KUKA KRL program: wkz_off_st_geo.src, wkz_off_st_geo.dat

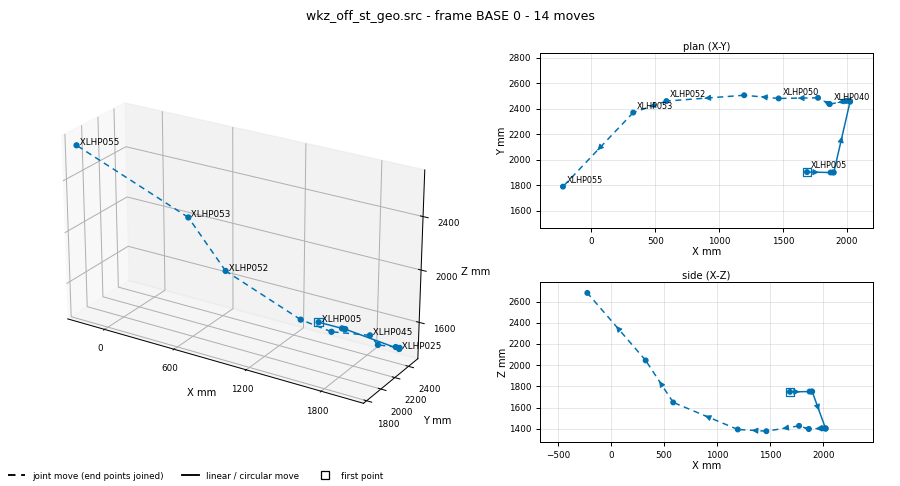
[picture p0: tool path of wkz_off_st_geo.src in frame BASE 0, 14 of 14 moves have a stored position in this frame; points joined in program order, loops and branches not executed]
--- wkz_off_st_geo.src ---
&ACCESS RVO2
&REL 409
&COMMENT Retira Gripper Geo
&PARAM DISKPATH = KRC:\R1\Program
DEF wkz_off_st_geo( )
;FOLD INI
   ;FOLD BASISTECH INI
      GLOBAL INTERRUPT DECL 3 WHEN $STOPMESS==TRUE DO IR_STOPM ( )
      INTERRUPT ON 3
      BAS (#INITMOV,0 )
   ;ENDFOLD (BASISTECH INI)
   ;FOLD SPOTTECH INI
      USERSPOT(#INIT)
   ;ENDFOLD (SPOTTECH INI)
   ;FOLD GRIPPERTECH INI
      USER_GRP(0,DUMMY,DUMMY,GDEFAULT)
   ;ENDFOLD (GRIPPERTECH INI)
   ;FOLD USER INI
      ;Make your modifications here

   ;ENDFOLD (USER INI)
;ENDFOLD (INI)

; Estacao P13.060 - Robo R1
; Programa: Pega Gripper Garra
; Accelo na Geobox. Gripper F5_6500_0026_656
; Caracterização dos meios de produção:
; 02/09/2014 09:15 Changes by KUKA Roboter do Brasil

chk_w8_wechs_ok ( )   ; CHECK FERRAMENTA: TOOL CHANGER

;FOLD OUT 3337 'R1_Retira Garra Geo' State=TRUE ;%{PE}%R 8.2.20,%MKUKATPBASIS,%COUT,%VOUTX,%P 2:3337, 3:R1_Retira Garra Geo, 5:TRUE, 6:
$OUT[3337]=TRUE
;ENDFOLD
;FOLD WAIT FOR ( IN 3337 'R1_Aguarda Lib. Entrar Geo' );%{PE}%R 8.2.20,%MKUKATPBASIS,%CEXT_WAIT_FOR,%VEXT_WAIT_FOR,%P 2:, 4:, 5:$IN, 6:3337, 7:R1_Aguarda Lib. Entrar Geo, 9:
WAIT FOR  ( $IN[3337] )
;ENDFOLD
;FOLD OUT 3337 'R1_Retira Garra Geo' State=FALSE ;%{PE}%R 8.2.20,%MKUKATPBASIS,%COUT,%VOUTX,%P 2:3337, 3:R1_Retira Garra Geo, 5:FALSE, 6:
$OUT[3337]=FALSE
;ENDFOLD
;FOLD OUT 3346 'R1_Entrega Peca Geo' State=FALSE ;%{PE}%R 8.2.20,%MKUKATPBASIS,%COUT,%VOUTX,%P 2:3346, 3:R1_Entrega Peca Geo, 5:FALSE, 6:
$OUT[3346]=FALSE
;ENDFOLD
;FOLD OUT 3343 'R1_Entregou Peca Geo' State=FALSE ;%{PE}%R 8.2.20,%MKUKATPBASIS,%COUT,%VOUTX,%P 2:3343, 3:R1_Entregou Peca Geo, 5:FALSE, 6:
$OUT[3343]=FALSE
;ENDFOLD

;FOLD OUT 3369 'Area de Solda' State=FALSE ;%{PE}%R 8.2.20,%MKUKATPBASIS,%COUT,%VOUTX,%P 2:3369, 3:Area de Solda, 5:FALSE, 6:
$OUT[3369]=FALSE
;ENDFOLD

;FOLD Kollision.Ueberwachung_3_Ein ;%{PE}%MKUKATPUSER
COLLSTOP( 3, 1 ) ;INTERRUPTUEBERWACHT
;ENDFOLD

;FOLD PTP LHP005 CONT Vel=60 % PDAT3 Tool[2]:Gripper Lat Esq Accelo Base[0];%{PE}%R 4.1.15,%MKUKATPBASIS,%CMOVE,%VPTP,%P 1:PTP, 2:LHP005, 3:C_PTP, 5:60, 7:PDAT3
$BWDSTART=FALSE
PDAT_ACT=PPDAT3
BAS (#PTP_DAT )
FDAT_ACT=FLHP005
BAS (#FRAMES )
BAS (#VEL_PTP,60 )
PTP  XLHP005 C_PTP
;ENDFOLD

;FOLD OUT 224 'Bloqueio MPS'  State= FALSE ;%{PE}%R 4.1.16,%MKUKATPBASIS,%COUT,%VOUTX,%P 2:224, 3:'Bloqueio MPS', 5:FALSE, 6:
$OUT[224]=FALSE
;ENDFOLD
;FOLD OUT 223 'Desbloqueio MPS'  State= TRUE ;%{PE}%R 4.1.16,%MKUKATPBASIS,%COUT,%VOUTX,%P 2:223, 3:'Desbloqueio MPS', 5:TRUE, 6:
$OUT[223]=TRUE
;ENDFOLD

;FOLD LIN LHP010 Vel=0.3 m/s CPDAT11 Tool[8]:Tool Changer Base[0];%{PE}%R 8.2.20,%MKUKATPBASIS,%CMOVE,%VLIN,%P 1:LIN, 2:LHP010, 3:, 5:0.3, 7:CPDAT11
$BWDSTART=FALSE
LDAT_ACT=LCPDAT11
FDAT_ACT=FLHP010
BAS(#CP_PARAMS,0.3)
LIN XLHP010
;ENDFOLD

;FOLD WAIT FOR IN 217 'MPS destravado'  State= TRUE ;%{PE}%R 4.1.16,%MKUKATPBASIS,%CWAIT_FOR,%VWAIT_FOR,%P 1:0, 2:217, 3:'MPS destravado', 5:TRUE, 6:
WAIT FOR $IN[217]==TRUE
;ENDFOLD
;FOLD WAIT FOR IN 221 'MPS travado'  State= FALSE ;%{PE}%R 4.1.16,%MKUKATPBASIS,%CWAIT_FOR,%VWAIT_FOR,%P 1:0, 2:221, 3:'MPS travado', 5:FALSE, 6:
WAIT FOR $IN[221]==FALSE
;ENDFOLD

;FOLD LIN LHP015 Vel=0.25 m/s CPDAT12 Tool[8]:Tool Changer Base[0];%{PE}%R 8.2.20,%MKUKATPBASIS,%CMOVE,%VLIN,%P 1:LIN, 2:LHP015, 3:, 5:0.25, 7:CPDAT12
$BWDSTART=FALSE
LDAT_ACT=LCPDAT12
FDAT_ACT=FLHP015
BAS(#CP_PARAMS,0.25)
LIN XLHP015
;ENDFOLD

;FOLD ;  posicao de pega do gripper;%{PE}%R 4.1.16,%MKUKATPBASIS,%CCOMMENT,%VNORMAL,%P 2: posicao de pega do gripper
;ENDFOLD
;FOLD LIN LHP020  Vel= 0.25 m/s CPDAT15 Tool[8]:Tool Changer Base[0];%{PE}%R 4.1.16,%MKUKATPBASIS,%CMOVE,%VLIN,%P 1:LIN, 2:LHP020, 3:, 5:0.25, 7:CPDAT15
$BWDSTART = FALSE
LDAT_ACT=LCPDAT15
BAS(#CP_DAT)
FDAT_ACT=FLHP020
BAS(#FRAMES)
BAS(#VEL_CP,0.25)
LIN XLHP020
;ENDFOLD

;FOLD WAIT Time= 1 sec;%{PE}%R 4.1.16,%MKUKATPBASIS,%CWAIT,%VWAIT,%P 2:1
WAIT SEC 1
;ENDFOLD
;FOLD WAIT FOR IN 219 'placas de suporte fundidas'  State= TRUE ;%{PE}%R 4.1.16,%MKUKATPBASIS,%CWAIT_FOR,%VWAIT_FOR,%P 1:0, 2:219, 3:'placas de suporte fundidas', 5:TRUE, 6:
WAIT FOR $IN[219]==TRUE
;ENDFOLD
;FOLD IBUS  OFF;%{PE}%R 4.1.16,%MKUKATPBASIS,%CIBUS,%VMAP,%P 2:#OFF, 3:1
$IBUS_OFF=$IBUS_ON
$IBUS_ON=0
;ENDFOLD
;FOLD OUT 223 'Desbloqueio MPS'  State= FALSE ;%{PE}%R 4.1.16,%MKUKATPBASIS,%COUT,%VOUTX,%P 2:223, 3:'Desbloqueio MPS', 5:FALSE, 6:
$OUT[223]=FALSE
;ENDFOLD
;FOLD OUT 224 'Bloqueio MPS'  State= TRUE ;%{PE}%R 4.1.16,%MKUKATPBASIS,%COUT,%VOUTX,%P 2:224, 3:'Bloqueio MPS', 5:TRUE, 6:
$OUT[224]=TRUE
;ENDFOLD
;FOLD WAIT FOR IN 217 'MPS destravado'  State= FALSE ;%{PE}%R 4.1.16,%MKUKATPBASIS,%CWAIT_FOR,%VWAIT_FOR,%P 1:0, 2:217, 3:'MPS destravado', 5:FALSE, 6:
WAIT FOR $IN[217]==FALSE
;ENDFOLD
;FOLD WAIT FOR IN 221 'MPS travado'  State= TRUE ;%{PE}%R 4.1.16,%MKUKATPBASIS,%CWAIT_FOR,%VWAIT_FOR,%P 1:0, 2:221, 3:'MPS travado', 5:TRUE, 6:
WAIT FOR $IN[221]==TRUE
;ENDFOLD
;FOLD IBUS  ON SEGMENT_2;%{PE}%R 4.1.16,%MKUKATPBASIS,%CIBUS,%VMAP,%P 2:#ON, 3:2
$IBUS_ON=IBUS_SEGMENT[2]
$IBUS_OFF=0
;ENDFOLD
;FOLD WAIT Time= 1 sec;%{PE}%R 4.1.16,%MKUKATPBASIS,%CWAIT,%VWAIT,%P 2:1
WAIT SEC 1
;ENDFOLD

;FOLD OUT 3366 'R1_Solicita Sair com Garra' State=TRUE ;%{PE}%R 8.2.20,%MKUKATPBASIS,%COUT,%VOUTX,%P 2:3366, 3:R1_Solicita Sair com Garra, 5:TRUE, 6:
$OUT[3366]=TRUE
;ENDFOLD
;FOLD WAIT FOR ( IN 3335 'R1_Aguarda Lib. Retirar Garra' );%{PE}%R 8.2.20,%MKUKATPBASIS,%CEXT_WAIT_FOR,%VEXT_WAIT_FOR,%P 2:, 4:, 5:$IN, 6:3335, 7:R1_Aguarda Lib. Retirar Garra, 9:
WAIT FOR  ( $IN[3335] )
;ENDFOLD
;FOLD OUT 3366 'R1_Solicita Sair com Garra' State=FALSE ;%{PE}%R 8.2.20,%MKUKATPBASIS,%COUT,%VOUTX,%P 2:3366, 3:R1_Solicita Sair com Garra, 5:FALSE, 6:
$OUT[3366]=FALSE
;ENDFOLD

;FOLD SET GRP 1  State= OPN  GDAT1;%{PE}%R 4.1.7,%MKUKATPGRP,%CGRP,%VGRP,%P 2:1, 4:1, 5:#NO, 6:GDAT1, 8:0, 10:0
H50(GRP,1,1,GGDAT1)
;ENDFOLD
chk_grp1_opn ( )
;FOLD OUT 4 'Liga Vacuo' State=FALSE ;%{PE}%R 8.2.20,%MKUKATPBASIS,%COUT,%VOUTX,%P 2:4, 3:Liga Vacuo, 5:FALSE, 6:
$OUT[4]=FALSE
;ENDFOLD
;FOLD PULSE 3 'Sopro' State=TRUE Time=2 sec;%{PE}%R 8.2.20,%MKUKATPBASIS,%COUT,%VPULSE,%P 2:3, 3:Sopro, 5:TRUE, 6:, 8:2
PULSE($OUT[3], TRUE,2)
;ENDFOLD
;FOLD PULSE 3335 'R1_Retirou Garra Geo' State=TRUE CONT Time=3 sec;%{PE}%R 8.2.20,%MKUKATPBASIS,%COUT,%VPULSE,%P 2:3335, 3:R1_Retirou Garra Geo, 5:TRUE, 6:CONTINUE, 8:3
CONTINUE
PULSE($OUT[3335], TRUE,3)
;ENDFOLD
;FOLD OUT 3369 'Area de Solda' State=TRUE ;%{PE}%R 8.2.20,%MKUKATPBASIS,%COUT,%VOUTX,%P 2:3369, 3:Area de Solda, 5:TRUE, 6:
$OUT[3369]=TRUE
;ENDFOLD

;FOLD LIN LHP025 CONT Vel= 0.2 m/s CPDAT5 Tool[2]:Gripper Lat Esq Accelo Base[0];%{PE}%R 4.1.16,%MKUKATPBASIS,%CMOVE,%VLIN,%P 1:LIN, 2:LHP025, 3:C_DIS, 5:0.2, 7:CPDAT5
$BWDSTART = FALSE
LDAT_ACT=LCPDAT5
BAS(#CP_DAT)
FDAT_ACT=FLHP025
BAS(#FRAMES)
BAS(#VEL_CP,0.2)
LIN XLHP025 C_DIS
;ENDFOLD
;FOLD LIN LHP030 CONT Vel= 0.3 m/s CPDAT3 Tool[2]:Gripper Lat Esq Accelo Base[0];%{PE}%R 4.1.16,%MKUKATPBASIS,%CMOVE,%VLIN,%P 1:LIN, 2:LHP030, 3:C_DIS, 5:0.3, 7:CPDAT3
$BWDSTART = FALSE
LDAT_ACT=LCPDAT3
BAS(#CP_DAT)
FDAT_ACT=FLHP030
BAS(#FRAMES)
BAS(#VEL_CP,0.3)
LIN XLHP030 C_DIS
;ENDFOLD

;FOLD LIN LHP035 CONT Vel=2 m/s CPDAT4 Tool[2]:Gripper Lat Esq Accelo Base[0];%{PE}%R 8.2.20,%MKUKATPBASIS,%CMOVE,%VLIN,%P 1:LIN, 2:LHP035, 3:C_DIS C_DIS, 5:2, 7:CPDAT4
$BWDSTART=FALSE
LDAT_ACT=LCPDAT4
FDAT_ACT=FLHP035
BAS(#CP_PARAMS,2)
LIN XLHP035 C_DIS C_DIS
;ENDFOLD
;FOLD WAIT FOR IN 219 'placas de suporte fundidas'  State= TRUE ;%{PE}%R 4.1.16,%MKUKATPBASIS,%CWAIT_FOR,%VWAIT_FOR,%P 1:0, 2:219, 3:'placas de suporte fundidas', 5:TRUE, 6:
WAIT FOR $IN[219]==TRUE
;ENDFOLD

;FOLD PTP LHP040 CONT Vel= 60 % P_OLP4 Tool[2]:Gripper Lat Esq Accelo Base[0];%{PE}%R 4.1.16,%MKUKATPBASIS,%CMOVE,%VPTP,%P 1:PTP, 2:LHP040, 3:C_PTP, 5:60, 7:P_OLP4
$BWDSTART = FALSE
PDAT_ACT=PP_OLP4
BAS(#PTP_DAT)
FDAT_ACT=FLHP040
BAS(#FRAMES)
BAS(#VEL_PTP,60)
PTP XLHP040 C_PTP
;ENDFOLD
;FOLD PTP LHP045 CONT Vel= 50 % PDAT26 Tool[2]:Gripper Lat Esq Accelo Base[0];%{PE}%R 4.1.16,%MKUKATPBASIS,%CMOVE,%VPTP,%P 1:PTP, 2:LHP045, 3:C_PTP, 5:50, 7:PDAT26
$BWDSTART = FALSE
PDAT_ACT=PPDAT26
BAS(#PTP_DAT)
FDAT_ACT=FLHP045
BAS(#FRAMES)
BAS(#VEL_PTP,50)
PTP XLHP045 C_PTP
;ENDFOLD
;FOLD PTP LHP050 CONT Vel=60 % PDAT11 Tool[2]:Gripper Lat Esq Accelo Base[0];%{PE}%R 8.2.20,%MKUKATPBASIS,%CMOVE,%VPTP,%P 1:PTP, 2:LHP050, 3:C_DIS, 5:60, 7:PDAT11
$BWDSTART=FALSE
PDAT_ACT=PPDAT11
FDAT_ACT=FLHP050
BAS(#PTP_PARAMS,60)
PTP XLHP050 C_DIS
;ENDFOLD
;FOLD PTP LHP051 CONT Vel=60 % PDAT7 Tool[2]:Gripper Lat Esq Accelo Base[0];%{PE}%R 8.2.20,%MKUKATPBASIS,%CMOVE,%VPTP,%P 1:PTP, 2:LHP051, 3:C_DIS, 5:60, 7:PDAT7
$BWDSTART=FALSE
PDAT_ACT=PPDAT7
FDAT_ACT=FLHP051
BAS(#PTP_PARAMS,60)
PTP XLHP051 C_DIS
;ENDFOLD
;FOLD PTP LHP052 CONT Vel=60 % PDAT10 Tool[2]:Gripper Lat Esq Accelo Base[0];%{PE}%R 8.2.20,%MKUKATPBASIS,%CMOVE,%VPTP,%P 1:PTP, 2:LHP052, 3:C_DIS, 5:60, 7:PDAT10
$BWDSTART=FALSE
PDAT_ACT=PPDAT10
FDAT_ACT=FLHP052
BAS(#PTP_PARAMS,60)
PTP XLHP052 C_DIS
;ENDFOLD
;FOLD PTP LHP053 CONT Vel=60 % PDAT9 Tool[2]:Gripper Lat Esq Accelo Base[0];%{PE}%R 8.2.20,%MKUKATPBASIS,%CMOVE,%VPTP,%P 1:PTP, 2:LHP053, 3:C_DIS, 5:60, 7:PDAT9
$BWDSTART=FALSE
PDAT_ACT=PPDAT9
FDAT_ACT=FLHP053
BAS(#PTP_PARAMS,60)
PTP XLHP053 C_DIS
;ENDFOLD
;FOLD PTP LHP055 CONT Vel=50 % PDAT22 Tool[2]:Gripper Lat Esq Accelo Base[0];%{PE}%R 8.2.20,%MKUKATPBASIS,%CMOVE,%VPTP,%P 1:PTP, 2:LHP055, 3:C_DIS, 5:50, 7:PDAT22
$BWDSTART=FALSE
PDAT_ACT=PPDAT22
FDAT_ACT=FLHP055
BAS(#PTP_PARAMS,50)
PTP XLHP055 C_DIS
;ENDFOLD

;FOLD OUT 3337 'R1_Retira Garra Geo' State=TRUE CONT;%{PE}%R 8.2.20,%MKUKATPBASIS,%COUT,%VOUTX,%P 2:3337, 3:R1_Retira Garra Geo, 5:TRUE, 6:CONTINUE
CONTINUE
$OUT[3337]=TRUE
;ENDFOLD

END

--- wkz_off_st_geo.dat ---
&ACCESS RVO2
&REL 409
&COMMENT Retira Gripper Geo
&PARAM DISKPATH = KRC:\R1\Program
DEFDAT  wkz_off_st_geo
;FOLD EXTERNAL DECLARATIONS;%{PE}%MKUKATPBASIS,%CEXT,%VCOMMON,%P
;FOLD GRIPPERTECH EXT
EXT  H50 (INT  :IN,INT  :IN,INT  :IN,GRP_TYP  :IN )
;ENDFOLD (GRIPPERTECH EXT)
;FOLD SPOTTECH EXT
EXT  USERSPOT (S_COMMAND  :IN,SPOT_TYPE  :IN )
;ENDFOLD (SPOTTECH EXT)
;FOLD BASISTECH EXT;%{PE}%MKUKATPBASIS,%CEXT,%VEXT,%P
EXT  BAS (BAS_COMMAND  :IN,REAL  :IN )
DECL INT SUCCESS
;ENDFOLD (BASISTECH EXT)
;FOLD USER EXT;%{E}%MKUKATPUSER,%CEXT,%VEXT,%P
;Make your modifications here

;ENDFOLD (USER EXT)
;ENDFOLD (EXTERNAL DECLARATIONS)

;# ============ START PATH : ba_p13060r1_ltc_01 =============
DECL FDAT FLHP020={TOOL_NO 8,BASE_NO 0,IPO_FRAME #BASE}
DECL E6POS XLHP020={X 1896.38098,Y 1901.17798,Z 1752.06396,A -85.0355911,B 75.0925217,C -86.0191422,S 18,T 35,E1 0.0,E2 0.0,E3 0.0,E4 0.0,E5 0.0,E6 0.0}
DECL FDAT Fp4={TOOL_NO 2,BASE_NO 0,IPO_FRAME #BASE}
DECL E6POS Xp4={X 1992.50098,Y 2460.31396,Z 1405.73596,A -89.0228882,B 0.185930401,C -89.5983276,S 2,T 35,E1 0.0,E2 0.0,E3 0.0,E4 0.0,E5 0.0,E6 0.0}
DECL LDAT LL_OLP2={VEL 0.25,ACC 90.0,APO_DIST 2.0,APO_FAC 0.0}
DECL FDAT FLHP040={TOOL_NO 2,BASE_NO 0,IPO_FRAME #BASE}
DECL PDAT PP_OLP4={VEL 100.0,ACC 90.0,APO_DIST 30.0}
DECL E6POS XLHP040={X 1864.59302,Y 2435.71997,Z 1398.99194,A -89.3946533,B 0.327209085,C -89.8916321,S 18,T 35,E1 0.0,E2 0.0,E3 0.0,E4 0.0,E5 0.0,E6 0.0}
DECL PDAT PPDAT3={VEL 60.0,ACC 85.0,APO_DIST 30.0}
DECL PDAT PPDAT4={VEL 100.0,ACC 90.0,APO_DIST 30.0,APO_MODE #CDIS}
DECL E6POS XLHP045={X 1772.84998,Y 2485.021,Z 1428.75696,A -89.6036911,B 5.70348883,C -90.1840286,S 18,T 35,E1 0.0,E2 0.0,E3 0.0,E4 0.0,E5 0.0,E6 0.0}
DECL FDAT FLHP045={TOOL_NO 2,BASE_NO 0,IPO_FRAME #BASE}
DECL E6POS XLHP050={X 1464.948,Y 2480.08301,Z 1378.42798,A -86.6316299,B 5.11988878,C -98.4016876,S 18,T 35,E1 0.0,E2 0.0,E3 0.0,E4 0.0,E5 0.0,E6 0.0}
DECL FDAT FLHP050={TOOL_NO 2,BASE_NO 0,IPO_FRAME #BASE}
DECL LDAT LCPDAT2={VEL 2.0,ACC 85.0,APO_DIST 20.0,APO_FAC 50.0}
DECL GRP_SUGG_T LAST_GRP={NUMBER[] "1                       ",STATE[] "1                       ",PARAMS[] "GDAT1                   "}
DECL GRP_TYP GGDAT1={G_APO #NO,GRP_TIME 0.200000003,CTRL #OFF,DLY 0,DST 1}
DECL E6POS XLHP025={X 2023.43896,Y 2454.15991,Z 1401.18994,A -89.1424637,B 0.328501195,C -89.5951538,S 18,T 35,E1 0.0,E2 0.0,E3 0.0,E4 0.0,E5 0.0,E6 0.0}
DECL FDAT FLHP025={TOOL_NO 2,BASE_NO 0,IPO_FRAME #BASE}
DECL LDAT LCPDAT5={VEL 2.0,ACC 100.0,APO_DIST 2.0,APO_FAC 50.0}
DECL E6POS XLHP030={X 2022.849,Y 2460.35303,Z 1406.90601,A -89.0257721,B 0.139669403,C -89.5021896,S 2,T 35,E1 0.0,E2 0.0,E3 0.0,E4 0.0,E5 0.0,E6 0.0}
DECL FDAT FLHP030={TOOL_NO 2,BASE_NO 0,IPO_FRAME #BASE}
DECL LDAT LCPDAT3={VEL 2.0,ACC 90.0,APO_DIST 2.0,APO_FAC 50.0}
DECL LDAT LCPDAT11={VEL 2.0,ACC 90.0,APO_DIST 100.0,APO_FAC 50.0}
DECL E6POS XLHP010={X 1871.48401,Y 1900.80396,Z 1751.72095,A -85.027832,B 75.0897369,C -86.0116425,S 18,T 35,E1 0.0,E2 0.0,E3 0.0,E4 0.0,E5 0.0,E6 0.0}
DECL FDAT FLHP010={TOOL_NO 8,BASE_NO 0,IPO_FRAME #BASE,TQ_STATE FALSE}
DECL E6POS XLHP055={X -221.914398,Y 1790.33997,Z 2680.93799,A -84.7821732,B 77.6812134,C -170.099701,S 18,T 43,E1 0.0,E2 0.0,E3 0.0,E4 0.0,E5 0.0,E6 0.0}
DECL FDAT FLHP055={TOOL_NO 2,BASE_NO 0,IPO_FRAME #BASE,TQ_STATE FALSE}
DECL PDAT PPDAT22={VEL 100.0,ACC 100.0,APO_DIST 10.0,APO_MODE #CDIS}
DECL LDAT LCPDAT12={VEL 2.0,ACC 75.0,APO_DIST 5.0,APO_FAC 50.0}
DECL PDAT PPDAT26={VEL 100.0,ACC 85.0,APO_DIST 30.0}
DECL E6POS XLHP015={X 1891.69495,Y 1901.10095,Z 1751.979,A -85.0317917,B 75.0909805,C -86.0155106,S 18,T 35,E1 0.0,E2 0.0,E3 0.0,E4 0.0,E5 0.0,E6 0.0}
DECL FDAT FLHP015={TOOL_NO 8,BASE_NO 0,IPO_FRAME #BASE,TQ_STATE FALSE}
DECL LDAT LCPDAT15={VEL 2.0,ACC 90.0,APO_DIST 100.0,APO_FAC 50.0}
DECL E6POS XLHP005={X 1686.87598,Y 1904.25806,Z 1748.90906,A -86.3585892,B 75.039093,C -87.1308594,S 2,T 35,E1 0.0,E2 0.0,E3 0.0,E4 0.0,E5 0.0,E6 0.0}
DECL FDAT FLHP005={TOOL_NO 8,BASE_NO 0,IPO_FRAME #BASE}
DECL BASIS_SUGG_T LAST_BASIS={POINT1[] "LHP052                  ",POINT2[] "LHP052                  ",CP_PARAMS[] "CPDAT0                  ",PTP_PARAMS[] "PDAT10                  ",CONT[] "                        ",CP_VEL[] "0.3                     ",PTP_VEL[] "60                      ",SYNC_PARAMS[] "SYNCDAT                 ",SPL_NAME[] "S0                      "}
DECL E6POS XLHP026={X 1779.83301,Y 2450.62012,Z 1399.65796,A -89.1403503,B 0.323707789,C -89.5841599,S 18,T 35,E1 0.0,E2 0.0,E3 0.0,E4 0.0,E5 0.0,E6 0.0}
DECL FDAT FLHP026={TOOL_NO 2,BASE_NO 0,IPO_FRAME #BASE,POINT2[] " ",TQ_STATE FALSE}
DECL LDAT LCPDAT1={VEL 2.0,ACC 100.0,APO_DIST 100.0,APO_FAC 50.0,AXIS_VEL 100.0,AXIS_ACC 100.0,ORI_TYP #VAR,CIRC_TYP #BASE,JERK_FAC 50.0,GEAR_JERK 50.0,EXAX_IGN 0}
DECL E6POS XLHP027={X 1762.18298,Y 2450.34692,Z 1381.23499,A -89.1904221,B 0.385173112,C -96.4581909,S 18,T 35,E1 0.0,E2 0.0,E3 0.0,E4 0.0,E5 0.0,E6 0.0}
DECL FDAT FLHP027={TOOL_NO 2,BASE_NO 0,IPO_FRAME #BASE,POINT2[] " ",TQ_STATE FALSE}
DECL PDAT PPDAT1={VEL 100.0,ACC 90.0,APO_DIST 100.0,GEAR_JERK 50.0}
DECL E6POS XLHP028={X 1762.04395,Y 2404.74902,Z 1375.10303,A -89.1892166,B 0.401495486,C -96.4518967,S 18,T 35,E1 0.0,E2 0.0,E3 0.0,E4 0.0,E5 0.0,E6 0.0}
DECL FDAT FLHP028={TOOL_NO 2,BASE_NO 0,IPO_FRAME #BASE,POINT2[] " ",TQ_STATE FALSE}
DECL PDAT PPDAT2={VEL 100.0,ACC 90.0,APO_DIST 100.0,GEAR_JERK 50.0}
DECL E6POS XLHP029={X 1651.26294,Y 2403.11597,Z 1374.71399,A -89.1894836,B 0.401636302,C -96.4478073,S 18,T 35,E1 0.0,E2 0.0,E3 0.0,E4 0.0,E5 0.0,E6 0.0}
DECL FDAT FLHP029={TOOL_NO 2,BASE_NO 0,IPO_FRAME #BASE,POINT2[] " ",TQ_STATE FALSE}
DECL PDAT PPDAT5={VEL 100.0,ACC 90.0,APO_DIST 100.0,GEAR_JERK 50.0}
DECL FDAT FLHP035={TOOL_NO 2,BASE_NO 0,IPO_FRAME #BASE,POINT2[] " ",TQ_STATE FALSE}
DECL E6POS XLHP035={X 1992.49902,Y 2460.31299,Z 1405.73401,A -89.0231323,B 0.186079606,C -89.5979233,S 18,T 35,E1 0.0,E2 0.0,E3 0.0,E4 0.0,E5 0.0,E6 0.0}
DECL LDAT LCPDAT4={VEL 2.0,ACC 90.0,APO_DIST 2.0,APO_FAC 50.0,AXIS_VEL 100.0,AXIS_ACC 100.0,ORI_TYP #VAR,CIRC_TYP #BASE,JERK_FAC 50.0,GEAR_JERK 50.0,EXAX_IGN 0}
DECL SPOT_SUGG_T LAST_SPOT={GUN[] " 1                      ",RETR_CMD[] "#OPN                    ",CHOISE[] "#FIRST                  ",CLO_TM[] "0                       ",PGNO1[] " 1                      ",PRESS1[] "0                       ",PGNO2[] " 1                      ",PRESS2[] "0                       ",SPOT_PARAMS[] "NORMAL                  "}
DECL E6POS XLHP036={X 1788.44397,Y 2466.40698,Z 1395.04797,A -89.6003494,B 0.3782776,C -89.9430923,S 18,T 35,E1 0.0,E2 0.0,E3 0.0,E4 0.0,E5 0.0,E6 0.0}
DECL FDAT FLHP036={TOOL_NO 2,BASE_NO 0,IPO_FRAME #BASE,POINT2[] " ",TQ_STATE FALSE}
DECL PDAT PPDAT6={VEL 100.0,ACC 90.0,APO_DIST 30.0,APO_MODE #CDIS,GEAR_JERK 50.0}
DECL LDAT LCPDAT6={VEL 2.0,ACC 90.0,APO_DIST 2.0,APO_FAC 50.0,AXIS_VEL 100.0,AXIS_ACC 100.0,ORI_TYP #VAR,CIRC_TYP #BASE,JERK_FAC 50.0,GEAR_JERK 50.0,EXAX_IGN 0}
DECL E6POS XLHP051={X 1195.36304,Y 2505.11108,Z 1394.828,A -83.3905563,B 11.3238802,C -106.139702,S 18,T 35,E1 0.0,E2 0.0,E3 0.0,E4 0.0,E5 0.0,E6 0.0}
DECL FDAT FLHP051={TOOL_NO 2,BASE_NO 0,IPO_FRAME #BASE,POINT2[] " ",TQ_STATE FALSE}
DECL PDAT PPDAT7={VEL 100.0,ACC 85.0,APO_DIST 100.0,APO_MODE #CDIS,GEAR_JERK 50.0}
DECL E6POS XLHP054={X 327.607391,Y 2369.56299,Z 2045.41394,A -78.953537,B 42.0104408,C -130.848007,S 18,T 35,E1 0.0,E2 0.0,E3 0.0,E4 0.0,E5 0.0,E6 0.0}
DECL FDAT FLHP054={TOOL_NO 2,BASE_NO 0,IPO_FRAME #BASE,POINT2[] " ",TQ_STATE FALSE}
DECL PDAT PPDAT8={VEL 100.0,ACC 85.0,APO_DIST 100.0,GEAR_JERK 50.0}
DECL E6POS XLHP053={X 327.606293,Y 2369.56494,Z 2045.42297,A -78.9541473,B 42.0112991,C -130.848801,S 18,T 35,E1 0.0,E2 0.0,E3 0.0,E4 0.0,E5 0.0,E6 0.0}
DECL FDAT FLHP053={TOOL_NO 2,BASE_NO 0,IPO_FRAME #BASE,POINT2[] " ",TQ_STATE FALSE}
DECL PDAT PPDAT9={VEL 100.0,ACC 85.0,APO_DIST 100.0,APO_MODE #CDIS,GEAR_JERK 50.0}
DECL E6POS XLHP052={X 586.967529,Y 2459.44604,Z 1649.63501,A -79.0598068,B 27.0512104,C -124.305901,S 18,T 35,E1 0.0,E2 0.0,E3 0.0,E4 0.0,E5 0.0,E6 0.0}
DECL FDAT FLHP052={TOOL_NO 2,BASE_NO 0,IPO_FRAME #BASE,POINT2[] " ",TQ_STATE FALSE}
DECL PDAT PPDAT10={VEL 100.0,ACC 85.0,APO_DIST 100.0,APO_MODE #CDIS,GEAR_JERK 50.0}
DECL PDAT PPDAT11={VEL 100.0,ACC 85.0,APO_DIST 30.0,APO_MODE #CDIS,GEAR_JERK 50.0}
ENDDAT
